screen "lgr_flujo" 1280x740
   Button "Botón_1" at 774,622 size 250x80; TextOff 'REGRESAR'
      on Click: ActivateScreen("controles flujo", 0)
   Button "Botón_3" at 211,622 size 250x80; TextOff 'TENDENCIAS'
      on Activate: ActivateScreen("tendencia lgr flujo", 0)
   Button "Botón_5" at 48,198 size 108x49; TextOff 'ON'
      on Click: InvertBit("on_lgr_flujo")
   Circle "Círculo_5" at 177,209 size 35x35
      Appearance <- "on_lgr_flujo"
   TextField "Campo de texto_1" at 41,278 size 99x25; Text 'SETPOINT'
   TextField "Campo de texto_2" at 75,333 size 135x25; Text 'CONSTANTES'
   TextField "Campo de texto_3" at 58,412 size 43x25; Text 'KP:'
   TextField "Campo de texto_4" at 59,471 size 34x25; Text 'KI:'
   TextField "Campo de texto_5" at 61,531 size 39x25; Text 'KD:'
   IOField "Campo ES_1" at 140,272 size 100x40; FormatPattern s999999999.999
      ProcessValue <- "ref_lgr_flujo"
   TextField "Campo de texto_6" at 42,85 size 191x25; Text 'CONTROL DE FLUJO'
   GraphicView "Visor de gráficos_7" at 499,243 size 138x216; Picture "Gráfico_11"
   GraphicView "Visor de gráficos_2" at 924,449 size 56x50; Picture "Gráfico_14"
   GraphicView "Visor de gráficos_3" at 554,448 size 53x52; Picture "Gráfico_15"
   GraphicView "Visor de gráficos_4" at 632,290 size 52x29; Picture "Gráfico_16"
   GraphicView "Visor de gráficos_9" at 381,509 size 123x85; Picture "Gráfico_19"
   GraphicView "Visor de gráficos_10" at 388,97 size 61x52; Picture "Gráfico_20"
   GraphicView "Visor de gráficos_11" at 525,67 size 33x57; Picture "Gráfico_21"
   GraphicView "Visor de gráficos_12" at 628,83 size 61x63; Picture "Gráfico_22"
   GraphicView "Visor de gráficos_15" at 681,256 size 62x64; Picture "Gráfico_23"
   GraphicView "Visor de gráficos_17" at 748,469 size 55x58; Picture "Gráfico_24"
   GraphicView "Visor de gráficos_18" at 739,263 size 53x56; Picture "Gráfico_25"
   GraphicView "Visor de gráficos_6" at 790,256 size 62x64; Picture "Gráfico_23"
   GraphicView "Visor de gráficos_19" at 850,290 size 52x29; Picture "Gráfico_16"
   GraphicView "Visor de gráficos_20" at 894,243 size 138x216; Picture "Gráfico_11"
   GraphicView "Visor de gráficos_21" at 603,471 size 92x29; Picture "Gráfico_16"
   GraphicView "Visor de gráficos_22" at 692,437 size 62x64; Picture "Gráfico_23"
   GraphicView "Visor de gráficos_24" at 801,437 size 62x64; Picture "Gráfico_23"
   GraphicView "Visor de gráficos_25" at 861,471 size 67x29; Picture "Gráfico_16"
   GraphicView "Visor de gráficos_1" at 734,515 size 56x50; Picture "Gráfico_14"
   GraphicView "Visor de gráficos_8" at 495,537 size 251x29; Picture "Gráfico_16"
   GraphicView "Visor de gráficos_13" at 306,490 size 54x52; Picture "Gráfico_15"
   GraphicView "Visor de gráficos_14" at 344,513 size 48x29; Picture "Gráfico_16"
   GraphicView "Visor de gráficos_16" at 353,115 size 38x29; Picture "Gráfico_16"
   GraphicView "Visor de gráficos_23" at 445,116 size 187x29; Picture "Gráfico_16"
   GraphicView "Visor de gráficos_26" at 435,221 size 46x68; Picture "Gráfico_26"
   GraphicView "Visor de gráficos_27" at 434,333 size 46x68; Picture "Gráfico_26"
   GraphicView "Visor de gráficos_28" at 462,279 size 45x10; Picture "Gráfico_16"
   GraphicView "Visor de gráficos_29" at 463,391 size 45x10; Picture "Gráfico_16"
   GraphicView "Visor de gráficos_30" at 304,155 size 31x344; Picture "Gráfico_17"
   GraphicView "Visor de gráficos_31" at 307,117 size 52x48; Picture "Gráfico_27"
   GraphicView "Visor de gráficos_32" at 683,116 size 60x29; Picture "Gráfico_16"
   GraphicView "Visor de gráficos_34" at 750,153 size 31x120; Picture "Gráfico_17"
   Bar "Barra_1" at 900,275 size 131x145; MinimumValue 0; MaximumValue 27000
      ProcessValue <- "Nivel tanque"
   GraphicView "Visor de gráficos_35" at 930,200 size 75x76; Picture "Gráfico_28"
   Circle "Círculo_6" at 647,144 size 23x23
      Appearance <- "d7"
   GraphicView "Visor de gráficos_37" at 282,217 size 80x80; Picture "Gráfico_30"
   Circle "Círculo_7" at 374,241 size 23x23
      Appearance <- "Activar Unidad Enfriadora"
   Circle "Círculo_8" at 379,403 size 23x23
      Appearance <- "Activar Unidad Calefactora"
   GraphicView "Visor de gráficos_36" at 282,365 size 80x80; Picture "Gráfico_31"
   Rectangle "Rectángulo_3" at 444,225 size 33x20
      Appearance <- "Switch de Nivel Alto Tanque 1 (NC)"
   Rectangle "Rectángulo_4" at 444,337 size 33x20
      Appearance <- "Switch de Nivel Bajo Tanque 1 (NO)"
   GraphicView "Visor de gráficos_5" at 1131,97 size 126x149; Picture "Gráfico_32"
   GraphicView "Visor de gráficos_33" at 1077,115 size 61x29; Picture "Gráfico_16"
   GraphicView "Visor de gráficos_38" at 1157,259 size 56x50; Picture "Gráfico_14"
   GraphicView "Visor de gráficos_39" at 1026,282 size 78x29; Picture "Gráfico_16"
   GraphicView "Visor de gráficos_40" at 1023,82 size 62x64; Picture "Gráfico_23"
   GraphicView "Visor de gráficos_41" at 1099,248 size 62x64; Picture "Gráfico_23"
   GraphicView "Visor de gráficos_42" at 1182,239 size 31x34; Picture "Gráfico_17"
   Circle "Círculo_9" at 1037,43 size 23x23
      Appearance <- "Abrir Valvula Llenado Tanque 3"
   GraphicView "Visor de gráficos_43" at 784,115 size 247x29; Picture "Gráfico_16"
   Circle "Círculo_10" at 1120,323 size 23x23
      Appearance <- "Abrir Valvula Vaciado Tanque 3"
   GraphicView "Visor de gráficos_44" at 739,117 size 53x53; Picture "Gráfico_34"
   GraphicView "Visor de gráficos_45" at 275,51 size 53x149; Picture "Gráfico_35"
   TextField "Campo de texto_9" at 123,12 size 125x25; Text 'Temperatura'
   TextField "Campo de texto_10" at 388,27 size 53x25; Text 'Flujo'
   TextField "Campo de texto_11" at 504,175 size 76x25; Text 'Presion'
   TextField "Campo de texto_12" at 560,10 size 201x25; Text 'Valvula Proporcional'
   TextField "Campo de texto_13" at 366,449 size 159x25; Text 'Velocidad Motor'
   TextField "Campo de texto_14" at 939,171 size 53x25; Text 'Nivel'
   IOField "Campo ES_3" at 613,42 size 96x32; FormatPattern s99999
      ProcessValue <- "valvula"
   IOField "Campo ES_4" at 492,145 size 96x32; FormatPattern s999999999.999
      ProcessValue <- "presion"
   IOField "Campo ES_5" at 379,56 size 96x32; FormatPattern s999999999.999
      ProcessValue <- "flujo"
   IOField "Campo ES_6" at 243,11 size 96x32; FormatPattern s999999999.999
      ProcessValue <- "temperatura"
   IOField "Campo ES_7" at 385,475 size 96x32; FormatPattern s99999
      ProcessValue <- "bomba"
   Button "Botón_6" at 680,251 size 61x79; TextOff 'Text'
      on Click: InvertBit("v1llen")
   Button "Botón_7" at 791,251 size 61x79; TextOff 'Text'
      on Click: InvertBit("v2llen")
   Button "Botón_8" at 1099,242 size 61x79; TextOff 'Text'
      on Click: InvertBit("v3")
   Button "Botón_9" at 1024,77 size 61x79; TextOff 'Text'
      on Click: InvertBit("v3 llen")
   Button "Botón_10" at 803,434 size 61x79; TextOff 'Text'
      on Click: InvertBit("v2vac")
   Button "Botón_11" at 694,431 size 61x79; TextOff 'Text'
      on Click: InvertBit("v1vac")
   Button "Botón_12" at 280,364 size 80x80; TextOff 'Text'
      on Click: InvertBit("calefactora")
   Button "Botón_13" at 282,217 size 80x80; TextOff 'Text'
      on Click: InvertBit("enfriadora")
   TextField "Campo de texto_7" at 72,357 size 142x25; Text 'DEL CONTROL'
   IOField "Campo ES_2" at 112,402 size 100x40; FormatPattern s999999999.999
      ProcessValue <- "kp_lgr_flujo"
   IOField "Campo ES_8" at 112,463 size 100x40; FormatPattern s999999999.999
      ProcessValue <- "ki_lgr_flujo"
   IOField "Campo ES_9" at 113,523 size 100x40; FormatPattern s999999999.999
      ProcessValue <- "kd_lgr_flujo"
   TextField "Campo de texto_8" at 36,110 size 238x25; Text 'LUGAR GEOMETRICO DE'
   TextField "Campo de texto_15" at 89,132 size 117x25; Text 'LAS RAICES'
   Circle "Círculo_1" at 712,405 size 23x23
      Appearance <- "Abrir Valvula Vaciado Tanque 1"
   Circle "Círculo_2" at 821,405 size 23x23
      Appearance <- "Abrir Valvula Vaciado Tanque 2"
   Circle "Círculo_3" at 700,227 size 23x23
      Appearance <- "Abrir Valvula Llenado Tanque 1"
   Circle "Círculo_4" at 809,225 size 23x23
      Appearance <- "Abrir Valvula Llenado Tanque 2"
   Button "Botón_4" at 1124,490 size 104x70; TextOff 'MANUAL'
      on Click: InvertBit("onproc")
   Button "Botón_14" at 383,511 size 120x84; TextOff 'Text'
      on Click: InvertBit("d7")

screen "tendencia lgr flujo" 1280x740
   Button "Botón_1" at 535,607 size 300x80; TextOff 'REGRESAR'
      on Click: ActivateScreen("lgr_flujo", 0)
   TrendView "Visor de curvas_1" at 164,122 size 991x414
   TextField "Campo de texto_1" at 276,63 size 722x39; Text 'TENDENCIA DEL CONTROL DE FLUJO POR LGR'

screen "sintonizacion presion" 1280x740
   Button "Botón_1" at 760,627 size 300x80; TextOff 'REGRESAR'
      on Click: ActivateScreen("controles presion", 0)
   GraphicView "Visor de gráficos_7" at 499,243 size 138x216; Picture "Gráfico_11"
   GraphicView "Visor de gráficos_2" at 924,449 size 56x50; Picture "Gráfico_14"
   GraphicView "Visor de gráficos_3" at 554,448 size 53x52; Picture "Gráfico_15"
   GraphicView "Visor de gráficos_4" at 632,290 size 52x29; Picture "Gráfico_16"
   GraphicView "Visor de gráficos_9" at 381,509 size 123x85; Picture "Gráfico_19"
   GraphicView "Visor de gráficos_10" at 388,97 size 61x52; Picture "Gráfico_20"
   GraphicView "Visor de gráficos_11" at 525,67 size 33x57; Picture "Gráfico_21"
   GraphicView "Visor de gráficos_12" at 628,83 size 61x63; Picture "Gráfico_22"
   GraphicView "Visor de gráficos_15" at 681,256 size 62x64; Picture "Gráfico_23"
   GraphicView "Visor de gráficos_17" at 748,469 size 55x58; Picture "Gráfico_24"
   GraphicView "Visor de gráficos_18" at 739,263 size 53x56; Picture "Gráfico_25"
   GraphicView "Visor de gráficos_6" at 790,256 size 62x64; Picture "Gráfico_23"
   GraphicView "Visor de gráficos_19" at 850,290 size 52x29; Picture "Gráfico_16"
   GraphicView "Visor de gráficos_20" at 894,243 size 138x216; Picture "Gráfico_11"
   GraphicView "Visor de gráficos_21" at 603,471 size 92x29; Picture "Gráfico_16"
   GraphicView "Visor de gráficos_22" at 692,437 size 62x64; Picture "Gráfico_23"
   GraphicView "Visor de gráficos_24" at 801,437 size 62x64; Picture "Gráfico_23"
   GraphicView "Visor de gráficos_25" at 861,471 size 67x29; Picture "Gráfico_16"
   GraphicView "Visor de gráficos_1" at 734,515 size 56x50; Picture "Gráfico_14"
   GraphicView "Visor de gráficos_8" at 495,537 size 251x29; Picture "Gráfico_16"
   GraphicView "Visor de gráficos_13" at 306,490 size 54x52; Picture "Gráfico_15"
   GraphicView "Visor de gráficos_14" at 344,513 size 48x29; Picture "Gráfico_16"
   GraphicView "Visor de gráficos_16" at 353,115 size 38x29; Picture "Gráfico_16"
   GraphicView "Visor de gráficos_23" at 445,116 size 187x29; Picture "Gráfico_16"
   GraphicView "Visor de gráficos_26" at 435,221 size 46x68; Picture "Gráfico_26"
   GraphicView "Visor de gráficos_27" at 434,333 size 46x68; Picture "Gráfico_26"
   GraphicView "Visor de gráficos_28" at 462,279 size 45x10; Picture "Gráfico_16"
   GraphicView "Visor de gráficos_29" at 463,391 size 45x10; Picture "Gráfico_16"
   GraphicView "Visor de gráficos_30" at 304,155 size 31x344; Picture "Gráfico_17"
   GraphicView "Visor de gráficos_31" at 307,117 size 52x48; Picture "Gráfico_27"
   GraphicView "Visor de gráficos_32" at 683,116 size 60x29; Picture "Gráfico_16"
   GraphicView "Visor de gráficos_34" at 750,153 size 31x120; Picture "Gráfico_17"
   IOField "Campo ES_1" at 398,477 size 96x32; FormatPattern s99999
      ProcessValue <- "bomba"
   IOField "Campo ES_2" at 370,54 size 96x32; FormatPattern s999999999.999
      ProcessValue <- "flujo"
   IOField "Campo ES_3" at 611,36 size 96x32; FormatPattern s99999
      ProcessValue <- "valvula"
   IOField "Campo ES_4" at 495,149 size 96x32; FormatPattern s999999999.999
      ProcessValue <- "presion"
   Bar "Barra_1" at 900,275 size 131x145; MinimumValue 0; MaximumValue 27000
      ProcessValue <- "Nivel tanque"
   GraphicView "Visor de gráficos_35" at 930,200 size 75x76; Picture "Gráfico_28"
   TextField "Campo de texto_1" at 31,256 size 99x25; Text 'SETPOINT'
   TextField "Campo de texto_2" at 59,340 size 135x25; Text 'CONSTANTES'
   TextField "Campo de texto_3" at 55,406 size 43x25; Text 'KP:'
   TextField "Campo de texto_4" at 57,454 size 40x25; Text 'KI:'
   TextField "Campo de texto_5" at 57,502 size 39x25; Text 'KD:'
   Button "Botón_6" at 680,251 size 61x79; TextOff 'Text'
      on Click: InvertBit("v1llen")
   Button "Botón_7" at 692,431 size 61x79; TextOff 'Text'
      on Click: InvertBit("v1vac")
   Button "Botón_8" at 792,253 size 61x79; TextOff 'Text'
      on Click: InvertBit("v2llen")
   Button "Botón_9" at 800,431 size 65x83; TextOff 'Text'
      on Click: InvertBit("v2vac")
   TextField "Campo de texto_6" at 40,81 size 216x25; Text 'CONTROL DE PRESION'
   TextField "Campo de texto_7" at 58,106 size 162x25; Text 'SINTONIZACION'
   IOField "Campo ES_6" at 137,251 size 100x40; FormatPattern s999999999.999
      ProcessValue <- "ref_sint_presion"
   Button "Botón_2" at 40,173 size 108x49; TextOff 'ON'
      on Click: InvertBit("on_sint_presion")
   Circle "Círculo_5" at 181,180 size 36x36
      Appearance <- "on_sint_presion"
   Circle "Círculo_6" at 647,144 size 23x23
      Appearance <- "d7"
   Button "Botón_3" at 166,625 size 300x80; TextOff 'TENDENCIAS'
      on Click: ActivateScreen("tendencia sintonizacion presion", 0)
   IOField "Campo ES_7" at 110,399 size 99x39; FormatPattern s999999999.999
      ProcessValue <- "kp_sint_pres"
   IOField "Campo ES_8" at 108,452 size 99x39; FormatPattern s999999999.999
      ProcessValue <- "ki_sint_presion"
   IOField "Campo ES_9" at 108,504 size 99x39; FormatPattern s999999999.999
      ProcessValue <- "kd_sint_presion"
   GraphicView "Visor de gráficos_37" at 282,217 size 80x80; Picture "Gráfico_30"
   Circle "Círculo_7" at 374,241 size 23x23
      Appearance <- "Activar Unidad Enfriadora"
   Circle "Círculo_8" at 379,403 size 23x23
      Appearance <- "Activar Unidad Calefactora"
   Button "Botón_5" at 280,216 size 82x80; TextOff 'Text'
      on Click: InvertBit("enfriadora")
   GraphicView "Visor de gráficos_36" at 282,365 size 80x80; Picture "Gráfico_31"
   Button "Botón_10" at 282,362 size 83x87; TextOff 'Text'
      on Click: InvertBit("calefactora")
   Rectangle "Rectángulo_2" at 444,225 size 33x20
      Appearance <- "Switch de Nivel Alto Tanque 1 (NC)"
   Rectangle "Rectángulo_4" at 444,337 size 33x20
      Appearance <- "Switch de Nivel Bajo Tanque 1 (NO)"
   TextField "Campo de texto_8" at 58,362 size 136x25; Text 'DEL CONTROL'
   GraphicView "Visor de gráficos_5" at 1131,97 size 126x149; Picture "Gráfico_32"
   GraphicView "Visor de gráficos_33" at 1077,115 size 61x29; Picture "Gráfico_16"
   GraphicView "Visor de gráficos_38" at 1157,259 size 56x50; Picture "Gráfico_14"
   GraphicView "Visor de gráficos_39" at 1026,282 size 78x29; Picture "Gráfico_16"
   GraphicView "Visor de gráficos_40" at 1023,82 size 62x64; Picture "Gráfico_23"
   GraphicView "Visor de gráficos_41" at 1099,248 size 62x64; Picture "Gráfico_23"
   GraphicView "Visor de gráficos_42" at 1182,239 size 31x34; Picture "Gráfico_17"
   Button "Botón_11" at 1024,76 size 61x79; TextOff 'Text'
      on Click: InvertBit("v3 llen")
   Button "Botón_12" at 1099,243 size 61x79; TextOff 'Text'
      on Click: InvertBit("v3")
   Circle "Círculo_9" at 1037,43 size 23x23
      Appearance <- "Abrir Valvula Llenado Tanque 3"
   GraphicView "Visor de gráficos_43" at 784,115 size 247x29; Picture "Gráfico_16"
   Circle "Círculo_10" at 1120,323 size 23x23
      Appearance <- "Abrir Valvula Vaciado Tanque 3"
   GraphicView "Visor de gráficos_44" at 739,117 size 53x53; Picture "Gráfico_34"
   GraphicView "Visor de gráficos_45" at 275,51 size 53x149; Picture "Gráfico_35"
   IOField "Campo ES_5" at 248,10 size 96x32; FormatPattern s999999999.999
      ProcessValue <- "temperatura"
   TextField "Campo de texto_9" at 123,12 size 125x25; Text 'Temperatura'
   TextField "Campo de texto_10" at 388,27 size 53x25; Text 'Flujo'
   TextField "Campo de texto_11" at 504,175 size 76x25; Text 'Presion'
   TextField "Campo de texto_12" at 560,10 size 201x25; Text 'Valvula Proporcional'
   TextField "Campo de texto_13" at 366,449 size 159x25; Text 'Velocidad Motor'
   TextField "Campo de texto_14" at 939,171 size 53x25; Text 'Nivel'
   Circle "Círculo_1" at 712,405 size 23x23
      Appearance <- "Abrir Valvula Vaciado Tanque 1"
   Circle "Círculo_2" at 821,405 size 23x23
      Appearance <- "Abrir Valvula Vaciado Tanque 2"
   Circle "Círculo_3" at 700,227 size 23x23
      Appearance <- "Abrir Valvula Llenado Tanque 1"
   Circle "Círculo_4" at 809,225 size 23x23
      Appearance <- "Abrir Valvula Llenado Tanque 2"
   Button "Botón_4" at 1124,490 size 104x70; TextOff 'MANUAL'
      on Click: InvertBit("onproc")
   Button "Botón_14" at 383,511 size 120x84; TextOff 'Text'
      on Click: InvertBit("d7")

screen "tendencia sintonizacion presion" 1280x740
   TrendView "Visor de curvas_1" at 200,122 size 918x394
   Button "Botón_1" at 509,614 size 300x80; TextOff 'REGRESAR'
      on Click: ActivateScreen("sintonizacion presion", 0)
   TextField "Campo de texto_1" at 234,48 size 971x39; Text 'TENDENCIA DEL CONTROL DE PRESION POR SINTONIZACION'

screen "fuzzy presion" 1280x740
   Button "Botón_1" at 914,622 size 250x80; TextOff 'REGRESAR'
      on Click: ActivateScreen("controles presion", 0)
   Button "Botón_2" at 118,622 size 250x80; TextOff 'PARAMETROS'
      on Click: ActivateScreen("parametros fuzzy presion", 0)
   Button "Botón_3" at 509,622 size 250x80; TextOff 'TENDENCIAS'
      on Click: ActivateScreen("tendencia fuzzy presion", 0)
   Button "Botón_5" at 43,193 size 108x49; TextOff 'ON'; TextOn 'OFF'
      on Click: InvertBit("onfuzz_presion")
   TextField "Campo de texto_1" at 33,269 size 99x25; Text 'SETPOINT'
   Circle "Círculo_6" at 167,202 size 32x32
      Appearance <- "onfuzz_presion"
   IOField "Campo ES_1" at 139,262 size 100x40; FormatPattern s999999999.999
      ProcessValue <- "reffuzz_presion"
   GraphicView "Visor de gráficos_7" at 499,243 size 138x216; Picture "Gráfico_11"
   GraphicView "Visor de gráficos_2" at 924,449 size 56x50; Picture "Gráfico_14"
   GraphicView "Visor de gráficos_3" at 554,448 size 53x52; Picture "Gráfico_15"
   GraphicView "Visor de gráficos_4" at 632,290 size 52x29; Picture "Gráfico_16"
   GraphicView "Visor de gráficos_9" at 381,509 size 123x85; Picture "Gráfico_19"
   GraphicView "Visor de gráficos_10" at 388,97 size 61x52; Picture "Gráfico_20"
   GraphicView "Visor de gráficos_11" at 525,67 size 33x57; Picture "Gráfico_21"
   GraphicView "Visor de gráficos_12" at 628,83 size 61x63; Picture "Gráfico_22"
   GraphicView "Visor de gráficos_15" at 681,256 size 62x64; Picture "Gráfico_23"
   GraphicView "Visor de gráficos_17" at 748,469 size 55x58; Picture "Gráfico_24"
   GraphicView "Visor de gráficos_18" at 739,263 size 53x56; Picture "Gráfico_25"
   GraphicView "Visor de gráficos_6" at 790,256 size 62x64; Picture "Gráfico_23"
   GraphicView "Visor de gráficos_19" at 850,290 size 52x29; Picture "Gráfico_16"
   GraphicView "Visor de gráficos_20" at 894,243 size 138x216; Picture "Gráfico_11"
   GraphicView "Visor de gráficos_21" at 603,471 size 92x29; Picture "Gráfico_16"
   GraphicView "Visor de gráficos_22" at 692,437 size 62x64; Picture "Gráfico_23"
   GraphicView "Visor de gráficos_24" at 801,437 size 62x64; Picture "Gráfico_23"
   GraphicView "Visor de gráficos_25" at 861,471 size 67x29; Picture "Gráfico_16"
   GraphicView "Visor de gráficos_1" at 734,515 size 56x50; Picture "Gráfico_14"
   GraphicView "Visor de gráficos_8" at 495,537 size 251x29; Picture "Gráfico_16"
   GraphicView "Visor de gráficos_13" at 306,490 size 54x52; Picture "Gráfico_15"
   GraphicView "Visor de gráficos_14" at 344,513 size 48x29; Picture "Gráfico_16"
   GraphicView "Visor de gráficos_16" at 353,115 size 38x29; Picture "Gráfico_16"
   GraphicView "Visor de gráficos_23" at 445,116 size 187x29; Picture "Gráfico_16"
   GraphicView "Visor de gráficos_26" at 435,221 size 46x68; Picture "Gráfico_26"
   GraphicView "Visor de gráficos_27" at 434,333 size 46x68; Picture "Gráfico_26"
   GraphicView "Visor de gráficos_28" at 462,279 size 45x10; Picture "Gráfico_16"
   GraphicView "Visor de gráficos_29" at 463,391 size 45x10; Picture "Gráfico_16"
   GraphicView "Visor de gráficos_30" at 304,155 size 31x344; Picture "Gráfico_17"
   GraphicView "Visor de gráficos_31" at 307,117 size 52x48; Picture "Gráfico_27"
   GraphicView "Visor de gráficos_32" at 683,116 size 60x29; Picture "Gráfico_16"
   GraphicView "Visor de gráficos_34" at 750,153 size 31x120; Picture "Gráfico_17"
   Bar "Barra_1" at 900,275 size 131x145; MinimumValue 0; MaximumValue 27000
      ProcessValue <- "Nivel tanque"
   GraphicView "Visor de gráficos_35" at 930,200 size 75x76; Picture "Gráfico_28"
   Circle "Círculo_5" at 647,144 size 23x23
      Appearance <- "d7"
   GraphicView "Visor de gráficos_37" at 282,217 size 80x80; Picture "Gráfico_30"
   Circle "Círculo_7" at 374,241 size 23x23
      Appearance <- "Activar Unidad Enfriadora"
   Circle "Círculo_8" at 379,403 size 23x23
      Appearance <- "Activar Unidad Calefactora"
   GraphicView "Visor de gráficos_36" at 282,365 size 80x80; Picture "Gráfico_31"
   Rectangle "Rectángulo_2" at 444,225 size 33x20
      Appearance <- "Switch de Nivel Alto Tanque 1 (NC)"
   Rectangle "Rectángulo_4" at 444,337 size 33x20
      Appearance <- "Switch de Nivel Bajo Tanque 1 (NO)"
   GraphicView "Visor de gráficos_5" at 1131,97 size 126x149; Picture "Gráfico_32"
   GraphicView "Visor de gráficos_33" at 1077,115 size 61x29; Picture "Gráfico_16"
   GraphicView "Visor de gráficos_38" at 1157,259 size 56x50; Picture "Gráfico_14"
   GraphicView "Visor de gráficos_39" at 1026,282 size 78x29; Picture "Gráfico_16"
   GraphicView "Visor de gráficos_40" at 1023,82 size 62x64; Picture "Gráfico_23"
   GraphicView "Visor de gráficos_41" at 1099,248 size 62x64; Picture "Gráfico_23"
   GraphicView "Visor de gráficos_42" at 1182,239 size 31x34; Picture "Gráfico_17"
   Circle "Círculo_9" at 1037,43 size 23x23
      Appearance <- "Abrir Valvula Llenado Tanque 3"
   GraphicView "Visor de gráficos_43" at 784,115 size 247x29; Picture "Gráfico_16"
   Circle "Círculo_10" at 1120,323 size 23x23
      Appearance <- "Abrir Valvula Vaciado Tanque 3"
   GraphicView "Visor de gráficos_44" at 739,117 size 53x53; Picture "Gráfico_34"
   GraphicView "Visor de gráficos_45" at 275,51 size 53x149; Picture "Gráfico_35"
   TextField "Campo de texto_9" at 123,12 size 125x25; Text 'Temperatura'
   TextField "Campo de texto_10" at 388,27 size 53x25; Text 'Flujo'
   TextField "Campo de texto_11" at 504,175 size 76x25; Text 'Presion'
   TextField "Campo de texto_12" at 560,10 size 201x25; Text 'Valvula Proporcional'
   TextField "Campo de texto_13" at 366,449 size 159x25; Text 'Velocidad Motor'
   TextField "Campo de texto_14" at 939,171 size 53x25; Text 'Nivel'
   IOField "Campo ES_3" at 249,15 size 96x32; FormatPattern s999999999.999
      ProcessValue <- "temperatura"
   IOField "Campo ES_4" at 371,58 size 96x32; FormatPattern s999999999.999
      ProcessValue <- "flujo"
   IOField "Campo ES_5" at 611,41 size 96x32; FormatPattern s99999
      ProcessValue <- "valvula"
   IOField "Campo ES_6" at 496,147 size 96x32; FormatPattern s999999999.999
      ProcessValue <- "presion"
   IOField "Campo ES_7" at 393,477 size 96x32; FormatPattern s99999
      ProcessValue <- "bomba"
   Button "Botón_6" at 1024,77 size 61x79; TextOff 'Text'
      on Click: InvertBit("v3 llen")
   Button "Botón_7" at 1101,244 size 61x79; TextOff 'Text'
      on Click: InvertBit("v3")
   Button "Botón_8" at 791,250 size 61x79; TextOff 'Text'
      on Click: InvertBit("v2llen")
   Button "Botón_9" at 681,252 size 61x79; TextOff 'Text'
      on Click: InvertBit("v1llen")
   Button "Botón_10" at 695,431 size 61x79; TextOff 'Text'
      on Click: InvertBit("v1vac")
   Button "Botón_11" at 802,431 size 61x79; TextOff 'Text'
      on Click: InvertBit("v2vac")
   Button "Botón_12" at 282,216 size 80x80; TextOff 'Text'
      on Click: InvertBit("enfriadora")
   Button "Botón_13" at 281,366 size 80x80; TextOff 'Text'
      on Click: InvertBit("calefactora")
   TextField "Campo de texto_6" at 41,91 size 216x25; Text 'CONTROL DE PRESION'
   TextField "Campo de texto_8" at 103,116 size 66x25; Text 'FUZZY'
   TextField "Campo de texto_2" at 69,333 size 133x25; Text 'PARAMETROS'
   TextField "Campo de texto_4" at 37,373 size 109x25; Text 'NEGATIVO'
   TextField "Campo de texto_5" at 78,424 size 55x25; Text 'CERO'
   TextField "Campo de texto_3" at 42,483 size 98x25; Text 'POSITIVO'
   IOField "Campo ES_2" at 138,366 size 100x40; FormatPattern s999999999.999
      ProcessValue <- "NEG_FUZZ_presion"
   IOField "Campo ES_8" at 138,417 size 100x40; FormatPattern s999999999.999
      ProcessValue <- "CERO_FUZ_presion"
   IOField "Campo ES_9" at 138,476 size 100x40; FormatPattern s999999999.999
      ProcessValue <- "POS_FUZZ_presion"
   TextField "Campo de texto_7" at 34,533 size 106x25; Text 'VARIADOR'
   IOField "Campo ES_10" at 138,526 size 100x40; FormatPattern s999999999.999
      ProcessValue <- "VARIADORFUZZ_presion"
   Circle "Círculo_1" at 712,405 size 23x23
      Appearance <- "Abrir Valvula Vaciado Tanque 1"
   Circle "Círculo_2" at 821,405 size 23x23
      Appearance <- "Abrir Valvula Vaciado Tanque 2"
   Circle "Círculo_3" at 700,227 size 23x23
      Appearance <- "Abrir Valvula Llenado Tanque 1"
   Circle "Círculo_4" at 809,225 size 23x23
      Appearance <- "Abrir Valvula Llenado Tanque 2"
   Button "Botón_4" at 1124,490 size 104x70; TextOff 'MANUAL'
      on Click: InvertBit("onproc")
   Button "Botón_14" at 383,511 size 120x84; TextOff 'Text'
      on Click: InvertBit("d7")

screen "tendencia fuzzy presion" 1280x740
   TextField "Campo de texto_1" at 311,49 size 736x39; Text 'TENDENCIA DEL CONTROL DE PRESION FUZZY'
   Button "Botón_1" at 509,611 size 300x80; TextOff 'REGRESAR'
      on Click: ActivateScreen("fuzzy presion", 0)
   TrendView "Visor de curvas_1" at 115,101 size 1088x445

screen "parametros fuzzy presion" 1280x740
   Button "Botón_1" at 1064,632 size 204x90; TextOff 'REGRESAR'
      on Click: ActivateScreen("fuzzy presion", 0)
   TextField "Campo de texto_1" at 511,104 size 253x25; Text 'UNIVERSOS DE DISCURSO'
   TextField "Campo de texto_2" at 346,157 size 69x25; Text 'ERROR'
   TextField "Campo de texto_3" at 785,157 size 216x25; Text 'DERIVADA DEL ERROR'
   TextField "Campo de texto_4" at 167,211 size 109x25; Text 'NEGATIVO'
   TextField "Campo de texto_5" at 208,262 size 55x25; Text 'CERO'
   TextField "Campo de texto_6" at 172,321 size 98x25; Text 'POSITIVO'
   TextField "Campo de texto_7" at 682,211 size 109x25; Text 'NEGATIVO'
   TextField "Campo de texto_8" at 723,262 size 55x25; Text 'CERO'
   TextField "Campo de texto_9" at 687,321 size 98x25; Text 'POSITIVO'
   IOField "Campo ES_1" at 272,203 size 80x40; FormatPattern s999999999.999
      ProcessValue <- "EN_1_presion"
   IOField "Campo ES_2" at 360,203 size 80x40; FormatPattern s999999999.999
      ProcessValue <- "EN_2_presion"
   IOField "Campo ES_3" at 448,203 size 80x40; FormatPattern s999999999.999
      ProcessValue <- "EN_3_presion"
   IOField "Campo ES_4" at 537,203 size 80x40; FormatPattern s999999999.999
      ProcessValue <- "EN_4_presion"
   IOField "Campo ES_5" at 272,255 size 80x40; FormatPattern s999999999.999
      ProcessValue <- "EZ_1_presion"
   IOField "Campo ES_6" at 360,255 size 80x40; FormatPattern s999999999.999
      ProcessValue <- "EZ_2_presion"
   IOField "Campo ES_7" at 448,255 size 80x40; FormatPattern s999999999.999
      ProcessValue <- "EZ_3_presion"
   IOField "Campo ES_8" at 537,255 size 80x40; FormatPattern s999999999.999
      ProcessValue <- "EZ_4_presion"
   IOField "Campo ES_9" at 272,314 size 80x40; FormatPattern s999999999.999
      ProcessValue <- "EP_1_presion"
   IOField "Campo ES_10" at 360,314 size 80x40; FormatPattern s999999999.999
      ProcessValue <- "EP_2_presion"
   IOField "Campo ES_11" at 448,314 size 80x40; FormatPattern s999999999.999
      ProcessValue <- "EP_3_presion"
   IOField "Campo ES_12" at 537,314 size 80x40; FormatPattern s999999999.999
      ProcessValue <- "EP_4_presion"
   IOField "Campo ES_13" at 793,203 size 80x40; FormatPattern s999999999.999
      ProcessValue <- "DEN_1_presion"
   IOField "Campo ES_14" at 884,203 size 80x40; FormatPattern s999999999.999
      ProcessValue <- "DEN_2_presion"
   IOField "Campo ES_15" at 971,203 size 80x40; FormatPattern s999999999.999
      ProcessValue <- "DEN_3_presion"
   IOField "Campo ES_16" at 1055,203 size 80x40; FormatPattern s999999999.999
      ProcessValue <- "DEN_4_presion"
   IOField "Campo ES_17" at 793,255 size 80x40; FormatPattern s999999999.999
      ProcessValue <- "DEZ_1_presion"
   IOField "Campo ES_18" at 793,314 size 80x40; FormatPattern s999999999.999
      ProcessValue <- "DEP_1_presion"
   IOField "Campo ES_19" at 884,255 size 80x40; FormatPattern s999999999.999
      ProcessValue <- "DEZ_2_presion"
   IOField "Campo ES_20" at 884,314 size 80x40; FormatPattern s999999999.999
      ProcessValue <- "DEP_2_presion"
   IOField "Campo ES_21" at 971,255 size 80x40; FormatPattern s999999999.999
      ProcessValue <- "DEZ_3_presion"
   IOField "Campo ES_22" at 971,314 size 80x40; FormatPattern s999999999.999
      ProcessValue <- "DEP_3_presion"
   IOField "Campo ES_23" at 1055,255 size 80x40; FormatPattern s999999999.999
      ProcessValue <- "DEZ_4_presion"
   IOField "Campo ES_24" at 1055,314 size 80x40; FormatPattern s999999999.999
      ProcessValue <- "DEP_4_presion"

screen "on-off peso" 1280x740
   TextField "Campo de texto_1" at 68,273 size 140x32; Text 'SETPOINT'
   TextField "Campo de texto_2" at 104,405 size 71x32; Text 'PESO'
   Button "Botón_1" at 48,183 size 108x49; TextOff 'ON'
      on Click: InvertBit("on_peso")
   IOField "Campo ES_1" at 51,313 size 176x58; FormatPattern s999999999.999
      ProcessValue <- "ref_onoff_peso"
   IOField "Campo ES_2" at 51,484 size 176x58; FormatPattern s999999999.999
      ProcessValue <- "peso tanque"
   Button "Botón_2" at 732,622 size 300x80; TextOff 'REGRESAR'
      on Click: ActivateScreen("controles peso", 0)
   GraphicView "Visor de gráficos_7" at 499,243 size 138x216; Picture "Gráfico_11"
   GraphicView "Visor de gráficos_2" at 924,449 size 56x50; Picture "Gráfico_14"
   GraphicView "Visor de gráficos_3" at 554,448 size 53x52; Picture "Gráfico_15"
   GraphicView "Visor de gráficos_4" at 632,290 size 52x29; Picture "Gráfico_16"
   GraphicView "Visor de gráficos_9" at 381,509 size 123x85; Picture "Gráfico_19"
   GraphicView "Visor de gráficos_10" at 388,97 size 61x52; Picture "Gráfico_20"
   GraphicView "Visor de gráficos_11" at 525,67 size 33x57; Picture "Gráfico_21"
   GraphicView "Visor de gráficos_12" at 628,83 size 61x63; Picture "Gráfico_22"
   GraphicView "Visor de gráficos_15" at 681,256 size 62x64; Picture "Gráfico_23"
   GraphicView "Visor de gráficos_17" at 748,469 size 55x58; Picture "Gráfico_24"
   GraphicView "Visor de gráficos_18" at 739,263 size 53x56; Picture "Gráfico_25"
   GraphicView "Visor de gráficos_6" at 790,256 size 62x64; Picture "Gráfico_23"
   GraphicView "Visor de gráficos_19" at 850,290 size 52x29; Picture "Gráfico_16"
   GraphicView "Visor de gráficos_20" at 894,243 size 138x216; Picture "Gráfico_11"
   GraphicView "Visor de gráficos_21" at 603,471 size 92x29; Picture "Gráfico_16"
   GraphicView "Visor de gráficos_22" at 692,437 size 62x64; Picture "Gráfico_23"
   GraphicView "Visor de gráficos_24" at 801,437 size 62x64; Picture "Gráfico_23"
   GraphicView "Visor de gráficos_25" at 861,471 size 67x29; Picture "Gráfico_16"
   GraphicView "Visor de gráficos_1" at 734,515 size 56x50; Picture "Gráfico_14"
   GraphicView "Visor de gráficos_8" at 495,537 size 251x29; Picture "Gráfico_16"
   GraphicView "Visor de gráficos_13" at 306,490 size 54x52; Picture "Gráfico_15"
   GraphicView "Visor de gráficos_14" at 344,513 size 48x29; Picture "Gráfico_16"
   GraphicView "Visor de gráficos_16" at 353,115 size 38x29; Picture "Gráfico_16"
   GraphicView "Visor de gráficos_23" at 445,116 size 187x29; Picture "Gráfico_16"
   GraphicView "Visor de gráficos_26" at 435,221 size 46x68; Picture "Gráfico_26"
   GraphicView "Visor de gráficos_27" at 434,333 size 46x68; Picture "Gráfico_26"
   GraphicView "Visor de gráficos_28" at 462,279 size 45x10; Picture "Gráfico_16"
   GraphicView "Visor de gráficos_29" at 463,391 size 45x10; Picture "Gráfico_16"
   GraphicView "Visor de gráficos_30" at 304,155 size 31x344; Picture "Gráfico_17"
   GraphicView "Visor de gráficos_31" at 307,117 size 52x48; Picture "Gráfico_27"
   GraphicView "Visor de gráficos_32" at 683,116 size 60x29; Picture "Gráfico_16"
   GraphicView "Visor de gráficos_34" at 750,153 size 31x120; Picture "Gráfico_17"
   Bar "Barra_1" at 900,275 size 131x145; MinimumValue 0; MaximumValue 27000
      ProcessValue <- "Nivel tanque"
   GraphicView "Visor de gráficos_35" at 930,200 size 75x76; Picture "Gráfico_28"
   Circle "Círculo_6" at 647,144 size 23x23
      Appearance <- "d7"
   GraphicView "Visor de gráficos_37" at 282,217 size 80x80; Picture "Gráfico_30"
   Circle "Círculo_7" at 374,241 size 23x23
      Appearance <- "Activar Unidad Enfriadora"
   Circle "Círculo_8" at 379,403 size 23x23
      Appearance <- "Activar Unidad Calefactora"
   GraphicView "Visor de gráficos_36" at 282,365 size 80x80; Picture "Gráfico_31"
   Rectangle "Rectángulo_2" at 444,225 size 33x20
      Appearance <- "Switch de Nivel Alto Tanque 1 (NC)"
   Rectangle "Rectángulo_4" at 444,337 size 33x20
      Appearance <- "Switch de Nivel Bajo Tanque 1 (NO)"
   GraphicView "Visor de gráficos_5" at 1131,97 size 126x149; Picture "Gráfico_32"
   GraphicView "Visor de gráficos_33" at 1077,115 size 61x29; Picture "Gráfico_16"
   GraphicView "Visor de gráficos_38" at 1157,259 size 56x50; Picture "Gráfico_14"
   GraphicView "Visor de gráficos_39" at 1026,282 size 78x29; Picture "Gráfico_16"
   GraphicView "Visor de gráficos_40" at 1023,82 size 62x64; Picture "Gráfico_23"
   GraphicView "Visor de gráficos_41" at 1099,248 size 62x64; Picture "Gráfico_23"
   GraphicView "Visor de gráficos_42" at 1182,239 size 31x34; Picture "Gráfico_17"
   Circle "Círculo_9" at 1037,43 size 23x23
      Appearance <- "Abrir Valvula Llenado Tanque 3"
   GraphicView "Visor de gráficos_43" at 784,115 size 247x29; Picture "Gráfico_16"
   Circle "Círculo_10" at 1120,323 size 23x23
      Appearance <- "Abrir Valvula Vaciado Tanque 3"
   GraphicView "Visor de gráficos_44" at 739,117 size 53x53; Picture "Gráfico_34"
   GraphicView "Visor de gráficos_45" at 275,51 size 53x149; Picture "Gráfico_35"
   TextField "Campo de texto_9" at 123,12 size 125x25; Text 'Temperatura'
   TextField "Campo de texto_10" at 388,27 size 53x25; Text 'Flujo'
   TextField "Campo de texto_11" at 504,175 size 76x25; Text 'Presion'
   TextField "Campo de texto_12" at 560,10 size 201x25; Text 'Valvula Proporcional'
   TextField "Campo de texto_13" at 366,449 size 159x25; Text 'Velocidad Motor'
   TextField "Campo de texto_14" at 939,171 size 53x25; Text 'Nivel'
   IOField "Campo ES_4" at 248,12 size 96x32; FormatPattern s999999999.999
      ProcessValue <- "temperatura"
   IOField "Campo ES_5" at 366,57 size 96x32; FormatPattern s999999999.999
      ProcessValue <- "flujo"
   IOField "Campo ES_6" at 608,40 size 96x32; FormatPattern s99999
      ProcessValue <- "valvula"
   IOField "Campo ES_7" at 395,476 size 96x32; FormatPattern s99999
      ProcessValue <- "bomba"
   Circle "Círculo_5" at 188,194 size 28x28
      Appearance <- "on_peso"
   IOField "Campo ES_8" at 500,147 size 96x32; FormatPattern s999999999.999
      ProcessValue <- "presion"
   Button "Botón_3" at 161,622 size 300x80; TextOff 'TENDENCIAS'
      on Click: ActivateScreen("tendencia on off peso", 0)
   TextField "Campo de texto_3" at 88,434 size 102x32; Text 'ACTUAL'
   TextField "Campo de texto_4" at 69,68 size 133x32; Text 'CONTROL'
   TextField "Campo de texto_5" at 100,98 size 71x32; Text 'PESO'
   TextField "Campo de texto_6" at 85,128 size 101x32; Text 'ON-OFF'
   Button "Botón_5" at 1024,75 size 61x79; TextOff 'Text'
      on Click: InvertBit("v3 llen")
   Button "Botón_6" at 1101,243 size 61x79; TextOff 'Text'
      on Click: InvertBit("v3")
   Button "Botón_7" at 681,251 size 61x79; TextOff 'Text'
      on Click: InvertBit("v1llen")
   Button "Botón_8" at 790,252 size 61x79; TextOff 'Text'
      on Click: InvertBit("v2llen")
   Button "Botón_9" at 803,433 size 61x79; TextOff 'Text'
      on Click: InvertBit("v2vac")
   Button "Botón_10" at 693,432 size 61x79; TextOff 'Text'
      on Click: InvertBit("v1vac")
   Button "Botón_11" at 282,365 size 80x80; TextOff 'Text'
      on Click: InvertBit("calefactora")
   Button "Botón_12" at 280,218 size 80x80; TextOff 'Text'
      on Click: InvertBit("enfriadora")
   Circle "Círculo_1" at 712,405 size 23x23
      Appearance <- "Abrir Valvula Vaciado Tanque 1"
   Circle "Círculo_2" at 821,405 size 23x23
      Appearance <- "Abrir Valvula Vaciado Tanque 2"
   Circle "Círculo_3" at 700,227 size 23x23
      Appearance <- "Abrir Valvula Llenado Tanque 1"
   Circle "Círculo_4" at 809,225 size 23x23
      Appearance <- "Abrir Valvula Llenado Tanque 2"
   Button "Botón_4" at 1124,490 size 104x70; TextOff 'MANUAL'
      on Click: InvertBit("onproc")
   Button "Botón_14" at 383,511 size 120x84; TextOff 'Text'
      on Click: InvertBit("d7")

screen "tendencia on off peso" 1280x740
   Button "Botón_1" at 509,615 size 300x80; TextOff 'REGRESAR'
      on Click: ActivateScreen("on-off peso", 0)
   TextField "Campo de texto_1" at 380,69 size 558x39; Text 'TENDENCIA DEL CONTROL DE PESO'
   TrendView "Visor de curvas_1" at 104,130 size 1122x414

screen "lgr nivel" 1280x740
   Button "Botón_1" at 792,623 size 250x80; TextOff 'REGRESAR'
      on Click: ActivateScreen("controles nivel", 0)
   Button "Botón_3" at 185,623 size 250x80; TextOff 'TENDENCIAS'
      on Click: ActivateScreen("tendencia lgr nivel", 0)
   Button "Botón_5" at 48,198 size 108x49; TextOff 'ON'
      on Click: InvertBit("on_lgr_nivel")
   Circle "Círculo_5" at 177,209 size 35x35
      Appearance <- "on_lgr_nivel"
   TextField "Campo de texto_1" at 41,278 size 99x25; Text 'SETPOINT'
   TextField "Campo de texto_2" at 75,333 size 135x25; Text 'CONSTANTES'
   TextField "Campo de texto_3" at 58,412 size 43x25; Text 'KP:'
   TextField "Campo de texto_4" at 59,471 size 34x25; Text 'KI:'
   TextField "Campo de texto_5" at 61,531 size 39x25; Text 'KD:'
   IOField "Campo ES_1" at 140,272 size 100x40; FormatPattern s999999999.999
      ProcessValue <- "ref_lgr_nivel"
   TextField "Campo de texto_6" at 42,85 size 188x25; Text 'CONTROL DE NIVEL'
   GraphicView "Visor de gráficos_7" at 499,243 size 138x216; Picture "Gráfico_11"
   GraphicView "Visor de gráficos_2" at 924,449 size 56x50; Picture "Gráfico_14"
   GraphicView "Visor de gráficos_3" at 554,448 size 53x52; Picture "Gráfico_15"
   GraphicView "Visor de gráficos_4" at 632,290 size 52x29; Picture "Gráfico_16"
   GraphicView "Visor de gráficos_9" at 381,509 size 123x85; Picture "Gráfico_19"
   GraphicView "Visor de gráficos_10" at 388,97 size 61x52; Picture "Gráfico_20"
   GraphicView "Visor de gráficos_11" at 525,67 size 33x57; Picture "Gráfico_21"
   GraphicView "Visor de gráficos_12" at 628,83 size 61x63; Picture "Gráfico_22"
   GraphicView "Visor de gráficos_15" at 681,256 size 62x64; Picture "Gráfico_23"
   GraphicView "Visor de gráficos_17" at 748,469 size 55x58; Picture "Gráfico_24"
   GraphicView "Visor de gráficos_18" at 739,263 size 53x56; Picture "Gráfico_25"
   GraphicView "Visor de gráficos_6" at 790,256 size 62x64; Picture "Gráfico_23"
   GraphicView "Visor de gráficos_19" at 850,290 size 52x29; Picture "Gráfico_16"
   GraphicView "Visor de gráficos_20" at 894,243 size 138x216; Picture "Gráfico_11"
   GraphicView "Visor de gráficos_21" at 603,471 size 92x29; Picture "Gráfico_16"
   GraphicView "Visor de gráficos_22" at 692,437 size 62x64; Picture "Gráfico_23"
   GraphicView "Visor de gráficos_24" at 801,437 size 62x64; Picture "Gráfico_23"
   GraphicView "Visor de gráficos_25" at 861,471 size 67x29; Picture "Gráfico_16"
   GraphicView "Visor de gráficos_1" at 734,515 size 56x50; Picture "Gráfico_14"
   GraphicView "Visor de gráficos_8" at 495,537 size 251x29; Picture "Gráfico_16"
   GraphicView "Visor de gráficos_13" at 306,490 size 54x52; Picture "Gráfico_15"
   GraphicView "Visor de gráficos_14" at 344,513 size 48x29; Picture "Gráfico_16"
   GraphicView "Visor de gráficos_16" at 353,115 size 38x29; Picture "Gráfico_16"
   GraphicView "Visor de gráficos_23" at 445,116 size 187x29; Picture "Gráfico_16"
   GraphicView "Visor de gráficos_26" at 435,221 size 46x68; Picture "Gráfico_26"
   GraphicView "Visor de gráficos_27" at 434,333 size 46x68; Picture "Gráfico_26"
   GraphicView "Visor de gráficos_28" at 462,279 size 45x10; Picture "Gráfico_16"
   GraphicView "Visor de gráficos_29" at 463,391 size 45x10; Picture "Gráfico_16"
   GraphicView "Visor de gráficos_30" at 304,155 size 31x344; Picture "Gráfico_17"
   GraphicView "Visor de gráficos_31" at 307,117 size 52x48; Picture "Gráfico_27"
   GraphicView "Visor de gráficos_32" at 683,116 size 60x29; Picture "Gráfico_16"
   GraphicView "Visor de gráficos_34" at 750,153 size 31x120; Picture "Gráfico_17"
   Bar "Barra_1" at 900,275 size 131x145; MinimumValue 0; MaximumValue 27000
      ProcessValue <- "Nivel tanque"
   GraphicView "Visor de gráficos_35" at 930,200 size 75x76; Picture "Gráfico_28"
   Circle "Círculo_6" at 647,144 size 23x23
      Appearance <- "d7"
   GraphicView "Visor de gráficos_37" at 282,217 size 80x80; Picture "Gráfico_30"
   Circle "Círculo_7" at 374,241 size 23x23
      Appearance <- "Activar Unidad Enfriadora"
   Circle "Círculo_8" at 379,403 size 23x23
      Appearance <- "Activar Unidad Calefactora"
   GraphicView "Visor de gráficos_36" at 282,365 size 80x80; Picture "Gráfico_31"
   Rectangle "Rectángulo_3" at 444,225 size 33x20
      Appearance <- "Switch de Nivel Alto Tanque 1 (NC)"
   Rectangle "Rectángulo_4" at 444,337 size 33x20
      Appearance <- "Switch de Nivel Bajo Tanque 1 (NO)"
   GraphicView "Visor de gráficos_5" at 1131,97 size 126x149; Picture "Gráfico_32"
   GraphicView "Visor de gráficos_33" at 1077,115 size 61x29; Picture "Gráfico_16"
   GraphicView "Visor de gráficos_38" at 1157,259 size 56x50; Picture "Gráfico_14"
   GraphicView "Visor de gráficos_39" at 1026,282 size 78x29; Picture "Gráfico_16"
   GraphicView "Visor de gráficos_40" at 1023,82 size 62x64; Picture "Gráfico_23"
   GraphicView "Visor de gráficos_41" at 1099,248 size 62x64; Picture "Gráfico_23"
   GraphicView "Visor de gráficos_42" at 1182,239 size 31x34; Picture "Gráfico_17"
   Circle "Círculo_9" at 1037,43 size 23x23
      Appearance <- "Abrir Valvula Llenado Tanque 3"
   GraphicView "Visor de gráficos_43" at 784,115 size 247x29; Picture "Gráfico_16"
   Circle "Círculo_10" at 1120,323 size 23x23
      Appearance <- "Abrir Valvula Vaciado Tanque 3"
   GraphicView "Visor de gráficos_44" at 739,117 size 53x53; Picture "Gráfico_34"
   GraphicView "Visor de gráficos_45" at 275,51 size 53x149; Picture "Gráfico_35"
   TextField "Campo de texto_9" at 123,12 size 125x25; Text 'Temperatura'
   TextField "Campo de texto_10" at 388,27 size 53x25; Text 'Flujo'
   TextField "Campo de texto_11" at 504,175 size 76x25; Text 'Presion'
   TextField "Campo de texto_12" at 560,10 size 201x25; Text 'Valvula Proporcional'
   TextField "Campo de texto_13" at 366,449 size 159x25; Text 'Velocidad Motor'
   TextField "Campo de texto_14" at 939,171 size 53x25; Text 'Nivel'
   IOField "Campo ES_3" at 613,42 size 96x32; FormatPattern s99999
      ProcessValue <- "valvula"
   IOField "Campo ES_4" at 492,145 size 96x32; FormatPattern s999999999.999
      ProcessValue <- "presion"
   IOField "Campo ES_5" at 379,56 size 96x32; FormatPattern s999999999.999
      ProcessValue <- "flujo"
   IOField "Campo ES_6" at 243,11 size 96x32; FormatPattern s999999999.999
      ProcessValue <- "temperatura"
   IOField "Campo ES_7" at 385,475 size 96x32; FormatPattern s99999
      ProcessValue <- "bomba"
   Button "Botón_6" at 680,251 size 61x79; TextOff 'Text'
      on Click: InvertBit("v1llen")
   Button "Botón_7" at 791,251 size 61x79; TextOff 'Text'
      on Click: InvertBit("v2llen")
   Button "Botón_8" at 1099,242 size 61x79; TextOff 'Text'
      on Click: InvertBit("v3")
   Button "Botón_9" at 1024,77 size 61x79; TextOff 'Text'
      on Click: InvertBit("v3 llen")
   Button "Botón_10" at 803,434 size 61x79; TextOff 'Text'
      on Click: InvertBit("v2vac")
   Button "Botón_11" at 694,431 size 61x79; TextOff 'Text'
      on Click: InvertBit("v1vac")
   Button "Botón_12" at 280,364 size 80x80; TextOff 'Text'
      on Click: InvertBit("calefactora")
   Button "Botón_13" at 282,217 size 80x80; TextOff 'Text'
      on Click: InvertBit("enfriadora")
   TextField "Campo de texto_7" at 72,357 size 142x25; Text 'DEL CONTROL'
   IOField "Campo ES_2" at 112,402 size 100x40; FormatPattern s999999999.999
      ProcessValue <- "kp_lgr_nivel"
   IOField "Campo ES_8" at 112,463 size 100x40; FormatPattern s999999999.999
      ProcessValue <- "ki_lgr_nivel"
   IOField "Campo ES_9" at 113,523 size 100x40; FormatPattern s999999999.999
      ProcessValue <- "kd_lgr_nivel"
   TextField "Campo de texto_8" at 36,110 size 238x25; Text 'LUGAR GEOMETRICO DE'
   TextField "Campo de texto_15" at 89,132 size 117x25; Text 'LAS RAICES'
   Circle "Círculo_1" at 712,405 size 23x23
      Appearance <- "Abrir Valvula Vaciado Tanque 1"
   Circle "Círculo_2" at 821,405 size 23x23
      Appearance <- "Abrir Valvula Vaciado Tanque 2"
   Circle "Círculo_3" at 700,227 size 23x23
      Appearance <- "Abrir Valvula Llenado Tanque 1"
   Circle "Círculo_4" at 809,225 size 23x23
      Appearance <- "Abrir Valvula Llenado Tanque 2"
   Button "Botón_4" at 1124,490 size 104x70; TextOff 'MANUAL'
      on Click: InvertBit("onproc")
   Button "Botón_14" at 383,511 size 120x84; TextOff 'Text'
      on Click: InvertBit("d7")

screen "on-off nivel" 1280x740
   TextField "Campo de texto_1" at 68,273 size 140x32; Text 'SETPOINT'
   TextField "Campo de texto_2" at 98,405 size 82x32; Text 'NIVEL'
   Button "Botón_1" at 48,183 size 108x49; TextOff 'ON'
      on Click: InvertBit("on_nivel")
   IOField "Campo ES_1" at 51,313 size 176x58; FormatPattern s999999999.999
      ProcessValue <- "ref_onoff_nivel"
   IOField "Campo ES_2" at 51,484 size 176x58; FormatPattern s999999999.999
      ProcessValue <- "nivel_tanque"
   Button "Botón_2" at 732,622 size 300x80; TextOff 'REGRESAR'
      on Click: ActivateScreen("controles nivel", 0)
   GraphicView "Visor de gráficos_7" at 499,243 size 138x216; Picture "Gráfico_11"
   GraphicView "Visor de gráficos_2" at 924,449 size 56x50; Picture "Gráfico_14"
   GraphicView "Visor de gráficos_3" at 554,448 size 53x52; Picture "Gráfico_15"
   GraphicView "Visor de gráficos_4" at 632,290 size 52x29; Picture "Gráfico_16"
   GraphicView "Visor de gráficos_9" at 381,509 size 123x85; Picture "Gráfico_19"
   GraphicView "Visor de gráficos_10" at 388,97 size 61x52; Picture "Gráfico_20"
   GraphicView "Visor de gráficos_11" at 525,67 size 33x57; Picture "Gráfico_21"
   GraphicView "Visor de gráficos_12" at 628,83 size 61x63; Picture "Gráfico_22"
   GraphicView "Visor de gráficos_15" at 681,256 size 62x64; Picture "Gráfico_23"
   GraphicView "Visor de gráficos_17" at 748,469 size 55x58; Picture "Gráfico_24"
   GraphicView "Visor de gráficos_18" at 739,263 size 53x56; Picture "Gráfico_25"
   GraphicView "Visor de gráficos_6" at 790,256 size 62x64; Picture "Gráfico_23"
   GraphicView "Visor de gráficos_19" at 850,290 size 52x29; Picture "Gráfico_16"
   GraphicView "Visor de gráficos_20" at 894,243 size 138x216; Picture "Gráfico_11"
   GraphicView "Visor de gráficos_21" at 603,471 size 92x29; Picture "Gráfico_16"
   GraphicView "Visor de gráficos_22" at 692,437 size 62x64; Picture "Gráfico_23"
   GraphicView "Visor de gráficos_24" at 801,437 size 62x64; Picture "Gráfico_23"
   GraphicView "Visor de gráficos_25" at 861,471 size 67x29; Picture "Gráfico_16"
   GraphicView "Visor de gráficos_1" at 734,515 size 56x50; Picture "Gráfico_14"
   GraphicView "Visor de gráficos_8" at 495,537 size 251x29; Picture "Gráfico_16"
   GraphicView "Visor de gráficos_13" at 306,490 size 54x52; Picture "Gráfico_15"
   GraphicView "Visor de gráficos_14" at 344,513 size 48x29; Picture "Gráfico_16"
   GraphicView "Visor de gráficos_16" at 353,115 size 38x29; Picture "Gráfico_16"
   GraphicView "Visor de gráficos_23" at 445,116 size 187x29; Picture "Gráfico_16"
   GraphicView "Visor de gráficos_26" at 435,221 size 46x68; Picture "Gráfico_26"
   GraphicView "Visor de gráficos_27" at 434,333 size 46x68; Picture "Gráfico_26"
   GraphicView "Visor de gráficos_28" at 462,279 size 45x10; Picture "Gráfico_16"
   GraphicView "Visor de gráficos_29" at 463,391 size 45x10; Picture "Gráfico_16"
   GraphicView "Visor de gráficos_30" at 304,155 size 31x344; Picture "Gráfico_17"
   GraphicView "Visor de gráficos_31" at 307,117 size 52x48; Picture "Gráfico_27"
   GraphicView "Visor de gráficos_32" at 683,116 size 60x29; Picture "Gráfico_16"
   GraphicView "Visor de gráficos_34" at 750,153 size 31x120; Picture "Gráfico_17"
   Bar "Barra_1" at 900,275 size 131x145; MinimumValue 0; MaximumValue 27000
      ProcessValue <- "Nivel tanque"
   GraphicView "Visor de gráficos_35" at 930,200 size 75x76; Picture "Gráfico_28"
   Circle "Círculo_6" at 647,144 size 23x23
      Appearance <- "d7"
   GraphicView "Visor de gráficos_37" at 282,217 size 80x80; Picture "Gráfico_30"
   Circle "Círculo_7" at 374,241 size 23x23
      Appearance <- "Activar Unidad Enfriadora"
   Circle "Círculo_8" at 379,403 size 23x23
      Appearance <- "Activar Unidad Calefactora"
   GraphicView "Visor de gráficos_36" at 282,365 size 80x80; Picture "Gráfico_31"
   Rectangle "Rectángulo_2" at 444,225 size 33x20
      Appearance <- "Switch de Nivel Alto Tanque 1 (NC)"
   Rectangle "Rectángulo_4" at 444,337 size 33x20
      Appearance <- "Switch de Nivel Bajo Tanque 1 (NO)"
   GraphicView "Visor de gráficos_5" at 1131,97 size 126x149; Picture "Gráfico_32"
   GraphicView "Visor de gráficos_33" at 1077,115 size 61x29; Picture "Gráfico_16"
   GraphicView "Visor de gráficos_38" at 1157,259 size 56x50; Picture "Gráfico_14"
   GraphicView "Visor de gráficos_39" at 1026,282 size 78x29; Picture "Gráfico_16"
   GraphicView "Visor de gráficos_40" at 1023,82 size 62x64; Picture "Gráfico_23"
   GraphicView "Visor de gráficos_41" at 1099,248 size 62x64; Picture "Gráfico_23"
   GraphicView "Visor de gráficos_42" at 1182,239 size 31x34; Picture "Gráfico_17"
   Circle "Círculo_9" at 1037,43 size 23x23
      Appearance <- "Abrir Valvula Llenado Tanque 3"
   GraphicView "Visor de gráficos_43" at 784,115 size 247x29; Picture "Gráfico_16"
   Circle "Círculo_10" at 1120,323 size 23x23
      Appearance <- "Abrir Valvula Vaciado Tanque 3"
   GraphicView "Visor de gráficos_44" at 739,117 size 53x53; Picture "Gráfico_34"
   GraphicView "Visor de gráficos_45" at 275,51 size 53x149; Picture "Gráfico_35"
   TextField "Campo de texto_9" at 123,12 size 125x25; Text 'Temperatura'
   TextField "Campo de texto_10" at 388,27 size 53x25; Text 'Flujo'
   TextField "Campo de texto_11" at 504,175 size 76x25; Text 'Presion'
   TextField "Campo de texto_12" at 560,10 size 201x25; Text 'Valvula Proporcional'
   TextField "Campo de texto_13" at 366,449 size 159x25; Text 'Velocidad Motor'
   TextField "Campo de texto_14" at 939,171 size 53x25; Text 'Nivel'
   IOField "Campo ES_4" at 248,12 size 96x32; FormatPattern s999999999.999
      ProcessValue <- "temperatura"
   IOField "Campo ES_5" at 366,57 size 96x32; FormatPattern s999999999.999
      ProcessValue <- "flujo"
   IOField "Campo ES_6" at 608,40 size 96x32; FormatPattern s99999
      ProcessValue <- "valvula"
   IOField "Campo ES_7" at 395,476 size 96x32; FormatPattern s99999
      ProcessValue <- "bomba"
   Circle "Círculo_5" at 188,194 size 28x28
      Appearance <- "on_nivel"
   IOField "Campo ES_8" at 500,147 size 96x32; FormatPattern s999999999.999
      ProcessValue <- "presion"
   Button "Botón_3" at 161,622 size 300x80; TextOff 'TENDENCIAS'
      on Click: ActivateScreen("tendencia on off nivel", 0)
   TextField "Campo de texto_3" at 88,434 size 102x32; Text 'ACTUAL'
   TextField "Campo de texto_4" at 69,68 size 133x32; Text 'CONTROL'
   TextField "Campo de texto_5" at 95,98 size 82x32; Text 'NIVEL'
   TextField "Campo de texto_6" at 85,128 size 101x32; Text 'ON-OFF'
   Button "Botón_5" at 1024,75 size 61x79; TextOff 'Text'
      on Click: InvertBit("v3 llen")
   Button "Botón_6" at 1101,243 size 61x79; TextOff 'Text'
      on Click: InvertBit("v3")
   Button "Botón_7" at 681,251 size 61x79; TextOff 'Text'
      on Click: InvertBit("v1llen")
   Button "Botón_8" at 790,252 size 61x79; TextOff 'Text'
      on Click: InvertBit("v2llen")
   Button "Botón_9" at 803,433 size 61x79; TextOff 'Text'
      on Click: InvertBit("v2vac")
   Button "Botón_10" at 693,432 size 61x79; TextOff 'Text'
      on Click: InvertBit("v1vac")
   Button "Botón_11" at 282,365 size 80x80; TextOff 'Text'
      on Click: InvertBit("calefactora")
   Button "Botón_12" at 280,218 size 80x80; TextOff 'Text'
      on Click: InvertBit("enfriadora")
   Circle "Círculo_1" at 712,405 size 23x23
      Appearance <- "Abrir Valvula Vaciado Tanque 1"
   Circle "Círculo_2" at 821,405 size 23x23
      Appearance <- "Abrir Valvula Vaciado Tanque 2"
   Circle "Círculo_3" at 700,227 size 23x23
      Appearance <- "Abrir Valvula Llenado Tanque 1"
   Circle "Círculo_4" at 809,225 size 23x23
      Appearance <- "Abrir Valvula Llenado Tanque 2"
   Button "Botón_4" at 1124,490 size 104x70; TextOff 'MANUAL'
      on Click: InvertBit("onproc")
   Button "Botón_14" at 383,511 size 120x84; TextOff 'Text'
      on Click: InvertBit("d7")

screen "tendencia on off nivel" 1280x740
   Button "Botón_1" at 509,615 size 300x80; TextOff 'REGRESAR'
      on Click: ActivateScreen("on-off nivel", 0)
   TextField "Campo de texto_1" at 380,69 size 573x39; Text 'TENDENCIA DEL CONTROL DE NIVEL'
   TrendView "Visor de curvas_1" at 108,126 size 1128x406

screen "tendencia lgr nivel" 1280x740
   Button "Botón_1" at 535,607 size 300x80; TextOff 'REGRESAR'
      on Click: ActivateScreen("lgr nivel", 0)
   TextField "Campo de texto_1" at 276,63 size 726x39; Text 'TENDENCIA DEL CONTROL DE NIVEL POR PID'
   TrendView "Visor de curvas_1" at 88,126 size 1148x418
*)